SUBAPPLICATION Uebung_021 (* Spiegelabfolge (1) *)
  (* Standard: 61499-2 *)
  (* Version 1.0, 2023-10-23, franz *)
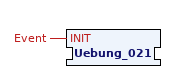
  EVENT_INPUT
    INIT;
  END_EVENT
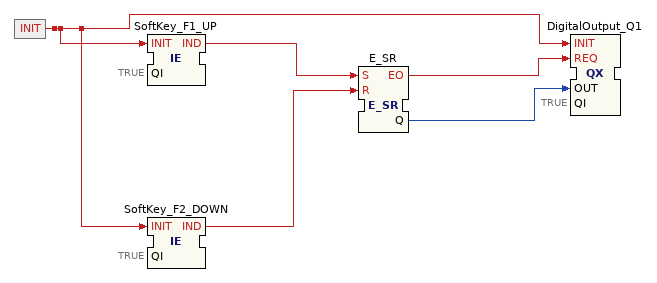
  (* START-Knopf *)
  (* Endlage &#10; *)
  FBS
    DigitalOutput_Q1 : QX(QI := TRUE);
    SoftKey_F1_UP : IE(QI := TRUE);
    E_SR : E_SR;
    SoftKey_F2_DOWN : IE(QI := TRUE);
  END_FBS
  EVENT_CONNECTIONS
    INIT TO SoftKey_F1_UP.INIT;
    INIT TO DigitalOutput_Q1.INIT;
    SoftKey_F1_UP.IND TO E_SR.S;
    INIT TO SoftKey_F2_DOWN.INIT;
    SoftKey_F2_DOWN.IND TO E_SR.R;
    E_SR.EO TO DigitalOutput_Q1.REQ;
  END_CONNECTIONS
  DATA_CONNECTIONS
    E_SR.Q TO DigitalOutput_Q1.OUT;
  END_CONNECTIONS
END_SUBAPPLICATION
